Omron CX-Programmer project NewProject (CX-Programmer 9.73)

# PLC NewPLC1: CP2E-N N

## Global symbols (name address type ; comment)
0 CHANNEL  ; MOTOR1
0.00 BOOL  ; LAMP 1
0.01 BOOL  ; BUTTON 1
0.02 BOOL  ; BUTTON2
0.03 BOOL  ; BUTTON3
100.00 BOOL  ; LAMP2
100.01 BOOL  ; DIR Motor1
100.02 BOOL  ; DIR1
100.03 BOOL  ; LAMP3
100.04 BOOL  ; BREAK1
100.05 BOOL  ; BREAK2
100.06 BOOL  ; EN1
100.07 BOOL  ; EN2
D0 CHANNEL  ; MOTOR2
D40 CHANNEL  ; INI M1
D50 CHANNEL  ; SAVE SET POINT
W0.00 BOOL  ; B_1
W0.01 BOOL  ; B_2
W0.02 BOOL  ; B_2
W0.03 BOOL  ; CW M1
W0.04 BOOL  ; CCW M1
W0.05 BOOL  ; BUTTON_SAVE
W0.06 BOOL  ; CW
W0.07 BOOL  ; CCW
W100.04 BOOL  ; Break2
W100.07 BOOL  ; EN2

## Program NewProgram1 (cyclic task 0)
Local symbols
HOME_M1 D80 UINT  ; Home Motor 1
HOME_M2 D81 UINT  ; Home Motor 2
POSITION D83 UINT  ; CORDINAT POSITION
SET_POINT D82 UINT  ; SET POINT TEACHING

### Section Set_Motor

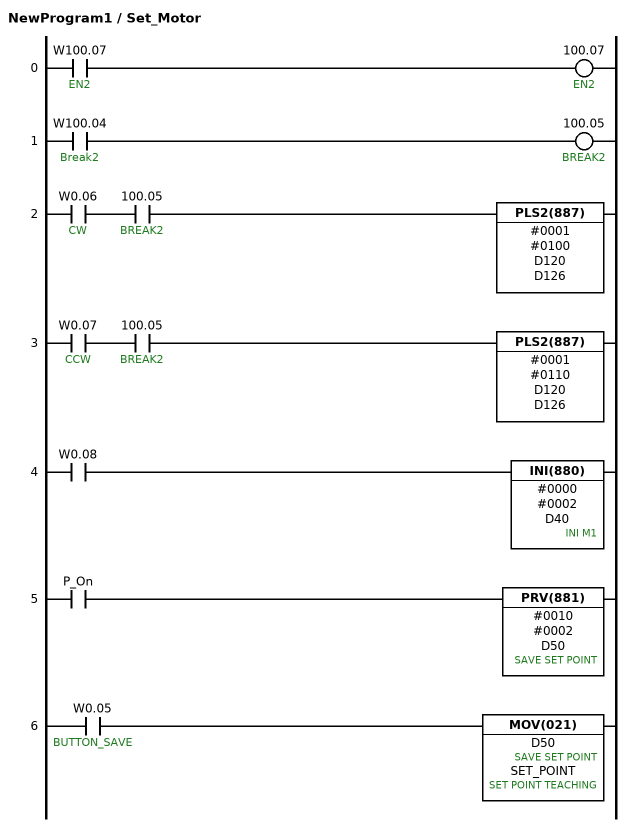
; rung 0
LD W100.07  ; EN2
OUT 100.07  ; EN2
; rung 1
LD W100.04  ; Break2
OUT 100.05  ; BREAK2
; rung 2
LD W0.06  ; CW
AND 100.05  ; BREAK2
PLS2(887) #0001 #0100 D120 D126
; rung 3
LD W0.07  ; CCW
AND 100.05  ; BREAK2
PLS2(887) #0001 #0110 D120 D126
; rung 4
LD W0.08
INI(880) #0000 #0002 D40  ; INI M1
; rung 5
LD P_On
PRV(881) #0010 #0002 D50  ; SAVE SET POINT
; rung 6
LD W0.05  ; BUTTON_SAVE
MOV(021) D50 SET_POINT  ; SAVE SET POINT, SET POINT TEACHING

### Section Section2

### Section Section3
; rung 0
END(001)

### Section End